PROGRAM MAIN
VAR
	enable AT%Q* : BOOL;
	speed AT%Q* : INT;
	motor_aan AT%Q* : INT;
	iSpeed : int;

	motor_bediening AT%Q* : BOOL;
	timer_tof: TOF;
	current_time: TIME;
	timer_ton: TON;
	
	blink: BOOL;
	blink_links: BOOL;
	blink_rechts: BOOL;
END_VAR

motor();

ACTION motor:
(*speed := 20000;

IF enable = TRUE THEN
	motor_aan := speed;
END_IF;*)

//enable := TRUE;
//speed := 20000;

	
(*timer_tof(IN:= enable, PT:= T#5S, Q=> motor_bediening, ET=> current_time);
	
IF current_time < T#2.5S
	THEN speed:= -20000;
END_IF;*)
	
timer_ton(IN:= NOT timer_ton.Q, PT:= T#10S);
blink_links := timer_ton.ET > T#5S;
blink_rechts := timer_ton.ET < T#5S;

motor_bediening := (enable AND blink_links) OR (enable AND blink_rechts);

IF timer_ton.ET < T#5S
	THEN speed:= iSpeed;
END_IF;
	
IF timer_ton.ET > T#5S
	THEN speed:= -iSpeed;
END_IF;
END_ACTION

END_PROGRAM

(* stored: Version 1.1.0.1, ProductVersion 3.1.4024.9
   POU MAIN: Id {73d23b6c-8b30-4588-8b3a-0edb20e25878}, SpecialFunc None
   Action motor: Id {cc3ce1ad-8f58-4bd2-ad22-b2c7c999bb6b} *)
